{attribute 'GeneratedUsingTerminal: CU2508-0000-0016'}
{attribute addProperty BoxType "CU2508-0000-0016"}
{attribute addProperty Id "EtcSlaveTerminalBaseInfoDataAT %I*InfoData_32EB74EA10"}
{attribute addProperty CRC "3667650902"}
{attribute addProperty Size "10"}
TYPE CU2508_DA9BE956 EXTENDS EtcSlaveTerminalBase :
STRUCT
	{attribute addProperty Name "InfoData"}
	InfoData : InfoData_32EB74EA;
END_STRUCT
END_TYPE

(* stored: Version 1.2.0.0, ProductVersion 3.1.4024.9
   DUT CU2508_DA9BE956: Id {a6ed83cf-b00d-4d86-8859-e969d4076138} *)
